ABB RAPID module: Module1.mod

MODULE Module1
	CONST robtarget Target_10:=[[380.00009573,-389.999758425,24.999857145],[-0.000000223,0.000000236,1,0.000000229],[-1,0,3,0],[9E+09,9E+09,9E+09,9E+09,9E+09,9E+09]];
	CONST robtarget Target_20:=[[380,370,25],[0,0,1,0],[0,0,0,0],[9E+09,9E+09,9E+09,9E+09,9E+09,9E+09]];
	CONST robtarget Target_30:=[[385,375,25],[0,0.707106781,0.707106781,0],[0,0,1,0],[9E+09,9E+09,9E+09,9E+09,9E+09,9E+09]];
	CONST robtarget Target_40:=[[390,370,25],[0,0.976296007,0.216439614,0],[0,0,2,0],[9E+09,9E+09,9E+09,9E+09,9E+09,9E+09]];
	CONST robtarget Target_50:=[[544.999847823,0,24.99966922],[0,1,0,-0.000000379],[0,0,2,0],[9E+09,9E+09,9E+09,9E+09,9E+09,9E+09]];
	PROC Path_10()
	    MoveL Target_10,v500,z50,tool0\WObj:=wobj0;
	    MoveL Target_20,v500,z50,tool0\WObj:=wobj0;
	ENDPROC
	PROC main()
	    Path_10;
	ENDPROC
ENDMODULE
